// TwinCAT 3 PLC project Knipperlicht
// ProgramVersion: 3.1.4024.0
// libraries:
//   Tc2_Standard, * (Beckhoff Automation GmbH)
//   Tc2_System, * (Beckhoff Automation GmbH)
//   Tc3_Module, * (Beckhoff Automation GmbH)
// project tree:
//   / PlcTask.TcTTO
//   POUs/ MAIN.TcPOU
// (motion and I/O tree: see PLC project trappenhuis_extraverlenging)
// real-time tasks:
//   TASK PlcTask: cycle T#10ms, priority 20, ADS port 350
//   TASK PlcTask1: cycle T#10ms, priority 21, ADS port 351
//   TASK PlcTask2: cycle T#10ms, priority 22, ADS port 352
//   TASK PlcTask3: cycle T#10ms, priority 23, ADS port 353
//   TASK PlcTask4: cycle T#10ms, priority 24, ADS port 354
//   TASK PlcTask5: cycle T#10ms, priority 25, ADS port 355
//   TASK PlcTask6: cycle T#10ms, priority 26, ADS port 356
//   TASK PlcTask7: cycle T#10ms, priority 27, ADS port 357
//   TASK PlcTask8: cycle T#10ms, priority 28, ADS port 358
//   TASK PlcTask9: cycle T#10ms, priority 29, ADS port 359
//   TASK PlcTask10: cycle T#10ms, priority 30, ADS port 360

CONFIGURATION Knipperlicht
    RESOURCE PLC ON TwinCAT3
        TASK PlcTask(INTERVAL := T#10ms, PRIORITY := 22);
        PROGRAM MAIN WITH PlcTask : MAIN;
    END_RESOURCE
END_CONFIGURATION

// ---- POUs/MAIN.TcPOU
PROGRAM MAIN
VAR
   fbBlinker1: TOF; // Timer voor lampje 1
   fbBlinker2: TOF; // Timer voor lampje 2
   nVoltage: REAL; // Ingangsspanning
   
   	Waarde: BYTE;
	potentiometer: INT;
   
   
	lamp1: BOOL;
	lamp2: BOOL;
END_VAR

(*
Knipperlicht (2 regels)

Schrijf een programma waarbij een lampje knippert aan een frequentie van 1 Hz – 50% Duty Cycle.

Uitbreiding: zorg dat de frequentie instelbaar is via de potentiometer met 500ms als minimum en 10s als maximum waarde.
 <br>Maak ook hier gebruik van de conversion operators. 

Uitbreiding: Ontwerp een knipperlamp met 4 verschillende knipperfrequenties.
De frequentie stijgt naarmate het analoge ingangsspanning vanuit de potentiometer stijgt. 
Bij een ingangsspanning lager dan 2V knippert het lampje met een frequentie van 0.5Hz,
tussen 2 en 4V 1 Hz, tussen 4 en 6V 2HZ en boven de 6V moeten er 2 lampjes om beurten knipperen met een frequentie van 5Hz.
*)
 
(*
Potentiometer inlezen en omzetten naar spanning (maximaal 2 regels)
*)
Waarde := LREAL_TO_BYTE(100 * (potentiometer / 32767.0)); // Scaled value from 0 to 100
nVoltage := (10.0 * potentiometer) / 32767.0; // Voltage value from 0V to 10V

IF nVoltage < 2 THEN
   fbBlinker1(IN:=NOT fbBlinker1.Q, PT:=T#1s); // 0.5 Hz
ELSIF nVoltage < 4 THEN
   fbBlinker1(IN:=NOT fbBlinker1.Q, PT:=T#500ms); // 1 Hz
ELSIF nVoltage < 6 THEN
   fbBlinker1(IN:=NOT fbBlinker1.Q, PT:=T#250ms); // 2 Hz
ELSE
   fbBlinker1(IN:=NOT fbBlinker1.Q, PT:=T#100ms); // 5 Hz voor lampje 1
   fbBlinker2(IN:=NOT fbBlinker2.Q, PT:=T#100ms); // 5 Hz voor lampje 2, alternerend
END_IF

lamp1 := fbBlinker1.Q;

lamp2 := (nVoltage >= 6) AND fbBlinker2.Q; // Lampje 2 enkel boven 6V

END_PROGRAM
